// TIA Portal project "TON_VS_P" (V15.1)

(* hardware
DEVICE "S71500/ET200MP station_1"  S7-1500 station
   slot 0: "Rail_0"  Rack  6ES7 590-1***0-0AA0
   slot 1: "PLC_1"  CPU 1513-1 PN  6ES7 513-1AL02-0AB0  V2.6
      slot 3: "CPU display_1"  6ES7591-1AA00-0AA0
DEVICE "HMI_1"  KTP900 Basic PN
   slot 0: "HMI_1"  KTP900 Basic PN  6AV2 123-2JB03-0AX0  15.1.0.0
   slot 1: "HMI_RT_1"  KTP900 Basic PN  6AV2 123-2JB03-0AX0  15.1.0.0
   slot 5: "HMI_1.IE_CP_1"  PROFINET Interface  15.0.1.0
      slot 1: "PROFINET Interface_1"  PROFINET Interface
         slot 1: "Port_1"  Port
*)

// ===== PLC "PLC_1"  CPU 1513-1 PN =====

VAR_GLOBAL   // PLC tag table "Default tag table"
   "Clock_Byte" AT %MB0 : Byte;
   "Clock_10Hz" AT %M0.0 : Bool;
   "Clock_5Hz" AT %M0.1 : Bool;
   "Clock_2.5Hz" AT %M0.2 : Bool;
   "Clock_2Hz" AT %M0.3 : Bool;
   "Clock_1.25Hz" AT %M0.4 : Bool;
   "Clock_1Hz" AT %M0.5 : Bool;
   "Clock_0.625Hz" AT %M0.6 : Bool;
   "Clock_0.5Hz" AT %M0.7 : Bool;
END_VAR

DATA_BLOCK "timer_ore_rfe_DB"   // DB1
{ S7_Optimized_Access := 'TRUE' }
VERSION : 0.1
// stored: InstanceOfName timer_ore_rfe
"timer_ore_rfe"
BEGIN
END_DATA_BLOCK

DATA_BLOCK "timer_ore_ton_DB"   // DB2
{ S7_Optimized_Access := 'TRUE' }
VERSION : 0.1
// stored: InstanceOfName timer_ore_ton
"timer_ore_ton"
BEGIN
END_DATA_BLOCK

DATA_BLOCK "timer_ton"   // DB3
{ S7_Optimized_Access := 'TRUE' }
VERSION : 0.1
   VAR
      btn_reset : Bool;
      permisiune_plecare : Bool;
      terminat : Bool;
      led_pornire : Bool;
      timer_s : Time;
      timer_m : USInt;
      timer_h : USInt;
      timer_s_secunde : Time;
   END_VAR
BEGIN
END_DATA_BLOCK

DATA_BLOCK "timer_rfe"   // DB4
{ S7_Optimized_Access := 'TRUE' }
VERSION : 0.1
   VAR
      btn_reset : Bool;
      permisiune_plecare : Bool;
      terminat : Bool;
      led_pornire : Bool;
      timer_s : USInt;
      timer_m : USInt;
      timer_h : USInt;
   END_VAR
BEGIN
END_DATA_BLOCK

// folder: System blocks/Program resources

DATA_BLOCK "timer_reset_rfe"   // DB5
{ S7_Optimized_Access := 'TRUE' }
AUTHOR : Simatic
FAMILY : IEC
NAME : IEC_TMR
VERSION : 1.0
// stored: InstanceOfName IEC_TIMER
"IEC_TIMER"
BEGIN
END_DATA_BLOCK

DATA_BLOCK "timer_reset_ton"   // DB6
{ S7_Optimized_Access := 'TRUE' }
AUTHOR : Simatic
FAMILY : IEC
NAME : IEC_TMR
VERSION : 1.0
// stored: InstanceOfName IEC_TIMER
"IEC_TIMER"
BEGIN
END_DATA_BLOCK

// folder: (top level)

FUNCTION_BLOCK "timer_ore_rfe"   // FB1, LAD
{ S7_Optimized_Access := 'TRUE' }
VERSION : 0.1
   VAR_INPUT
      reset : Bool;
   END_VAR
   VAR_OUTPUT
      terminat : Bool;
   END_VAR
   VAR_IN_OUT
      permisiune_plecare : Bool;
      timer_s : USInt;
      timer_m : USInt;
      timer_h : USInt;
   END_VAR
   VAR
      re1 : Bool;
   END_VAR
   VAR_TEMP   // added for the SCL form of the ladder/FBD networks
      _w1 : Bool;
   END_VAR
BEGIN

REGION Network 1: timer secunde
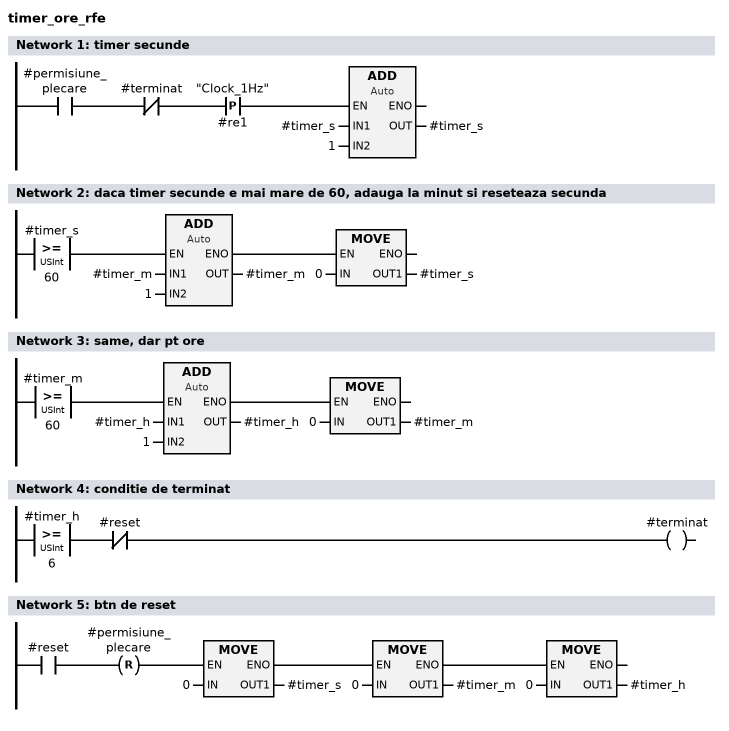
   RUNG wire#powerrail
      Contact( #permisiune_plecare )
      I_Contact( #terminat )
      P_Contact(operand := "Clock_1Hz", bit := #re1)
      Add(in1 := #timer_s, in2 := 1, out => #timer_s)
   END_RUNG
   // the same network as SCL:
   #_w1 := #permisiune_plecare AND NOT #terminat AND "Clock_1Hz" AND NOT #re1;   // rising edge of "Clock_1Hz"
   #re1 := "Clock_1Hz";
   IF #_w1 THEN #timer_s := #timer_s + 1; END_IF;
END_REGION

REGION Network 2: daca timer secunde e mai mare de 60, adauga la minut si reseteaza secunda
   RUNG wire#powerrail
      { S7_Templates := "SrcType := USInt" } GE_Contact(in1 := #timer_s, in2 := 60)
      Add(in1 := #timer_m, in2 := 1, out => #timer_m)
      Move(in := 0, out1 => #timer_s)
   END_RUNG
   // the same network as SCL:
   IF #timer_s >= 60 THEN
       #timer_m := #timer_m + 1;
       #timer_s := 0;
   END_IF;
END_REGION

REGION Network 3: same, dar pt ore
   RUNG wire#powerrail
      { S7_Templates := "SrcType := USInt" } GE_Contact(in1 := #timer_m, in2 := 60)
      Add(in1 := #timer_h, in2 := 1, out => #timer_h)
      Move(in := 0, out1 => #timer_m)
   END_RUNG
   // the same network as SCL:
   IF #timer_m >= 60 THEN
       #timer_h := #timer_h + 1;
       #timer_m := 0;
   END_IF;
END_REGION

REGION Network 4: conditie de terminat
   RUNG wire#powerrail
      { S7_Templates := "SrcType := USInt" } GE_Contact(in1 := #timer_h, in2 := 6)
      I_Contact( #reset )
      Coil( #terminat )
   END_RUNG
   // the same network as SCL:
   #terminat := (#timer_h >= 6) AND NOT #reset;
END_REGION

REGION Network 5: btn de reset
   RUNG wire#powerrail
      Contact( #reset )
      R_Coil( #permisiune_plecare )
      Move(in := 0, out1 => #timer_s)
      Move(in := 0, out1 => #timer_m)
      Move(in := 0, out1 => #timer_h)
   END_RUNG
   // the same network as SCL:
   IF #reset THEN
       #permisiune_plecare := FALSE;
       #timer_s := 0;
       #timer_m := 0;
       #timer_h := 0;
   END_IF;
END_REGION
END_FUNCTION_BLOCK

FUNCTION_BLOCK "timer_ore_ton"   // FB2, LAD
TITLE = aceasta functie nu prea o sa aiba sens, but bare with me ig
{ S7_Optimized_Access := 'TRUE' }
VERSION : 0.1
   VAR_INPUT
      reset : Bool;
   END_VAR
   VAR_OUTPUT
      terminat : Bool;
   END_VAR
   VAR_IN_OUT
      permisiune_plecare : Bool;
      time_ore : USInt;
      time_min : USInt;
      time_sec : Time;
   END_VAR
   VAR
      ton_s : TON_TIME;
      ton_aux : TON_TIME;
      terminat_secunde : Bool;
      plecare_sec : Bool;
      plecare_min : Bool;
      re1 : Bool;
      plecare_ora : Bool;
      adaugat_minut : Bool;
   END_VAR
   VAR_TEMP   // added for the SCL form of the ladder/FBD networks
      _w1 : Bool;
   END_VAR
BEGIN

REGION Network 1
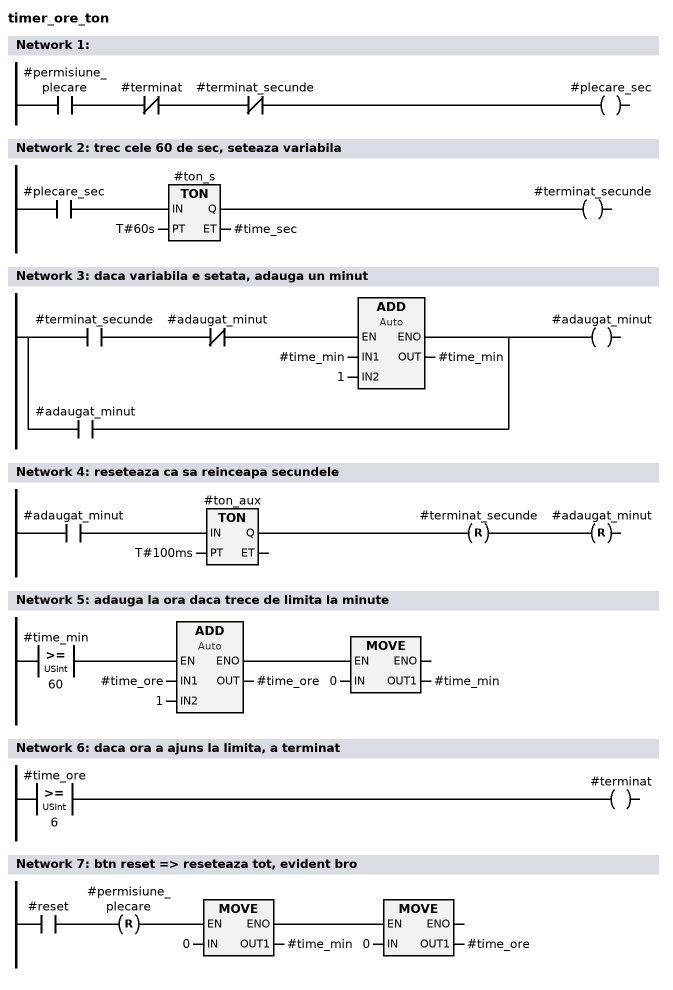
   RUNG wire#powerrail
      Contact( #permisiune_plecare )
      I_Contact( #terminat )
      I_Contact( #terminat_secunde )
      Coil( #plecare_sec )
   END_RUNG
   // the same network as SCL:
   #plecare_sec := #permisiune_plecare AND NOT #terminat AND NOT #terminat_secunde;
END_REGION

REGION Network 2: trec cele 60 de sec, seteaza variabila
   #ton_s(IN := #plecare_sec, PT := T#60s, ET => #time_sec);   // TON
   #terminat_secunde := #ton_s.Q;
END_REGION

REGION Network 3: daca variabila e setata, adauga un minut
   RUNG wire#powerrail
      Contact( #terminat_secunde )
      I_Contact( #adaugat_minut )
      Add(in1 := #time_min, in2 := 1, out => #time_min)
      wire#w1
      Coil( #adaugat_minut )
   END_RUNG
   RUNG wire#powerrail
      Contact( #adaugat_minut )
   END_RUNG wire#w1
   // the same network as SCL:
   #_w1 := #terminat_secunde AND NOT #adaugat_minut;
   IF #_w1 THEN #time_min := #time_min + 1; END_IF;
   #adaugat_minut := #_w1 OR #adaugat_minut;
END_REGION

REGION Network 4: reseteaza ca sa reinceapa secundele
   #ton_aux(IN := #adaugat_minut, PT := T#100ms);   // TON
   IF #ton_aux.Q THEN
       #terminat_secunde := FALSE;
       #adaugat_minut := FALSE;
   END_IF;
END_REGION

REGION Network 5: adauga la ora daca trece de limita la minute
   RUNG wire#powerrail
      { S7_Templates := "SrcType := USInt" } GE_Contact(in1 := #time_min, in2 := 60)
      Add(in1 := #time_ore, in2 := 1, out => #time_ore)
      Move(in := 0, out1 => #time_min)
   END_RUNG
   // the same network as SCL:
   IF #time_min >= 60 THEN
       #time_ore := #time_ore + 1;
       #time_min := 0;
   END_IF;
END_REGION

REGION Network 6: daca ora a ajuns la limita, a terminat
   RUNG wire#powerrail
      { S7_Templates := "SrcType := USInt" } GE_Contact(in1 := #time_ore, in2 := 6)
      Coil( #terminat )
   END_RUNG
   // the same network as SCL:
   #terminat := #time_ore >= 6;
END_REGION

REGION Network 7: btn reset => reseteaza tot, evident bro
   RUNG wire#powerrail
      Contact( #reset )
      R_Coil( #permisiune_plecare )
      Move(in := 0, out1 => #time_min)
      Move(in := 0, out1 => #time_ore)
   END_RUNG
   // the same network as SCL:
   IF #reset THEN
       #permisiune_plecare := FALSE;
       #time_min := 0;
       #time_ore := 0;
   END_IF;
END_REGION
END_FUNCTION_BLOCK

ORGANIZATION_BLOCK "Main"   // OB1, LAD, ProgramCycle
TITLE = "Main Program Sweep (Cycle)"
{ S7_Optimized_Access := 'TRUE' }
VERSION : 0.1
   VAR_INPUT
      Initial_Call : Bool;   // Initial call of this OB
      Remanence : Bool;   // =True, if remanent data are available
   END_VAR
BEGIN

REGION Network 1: functii
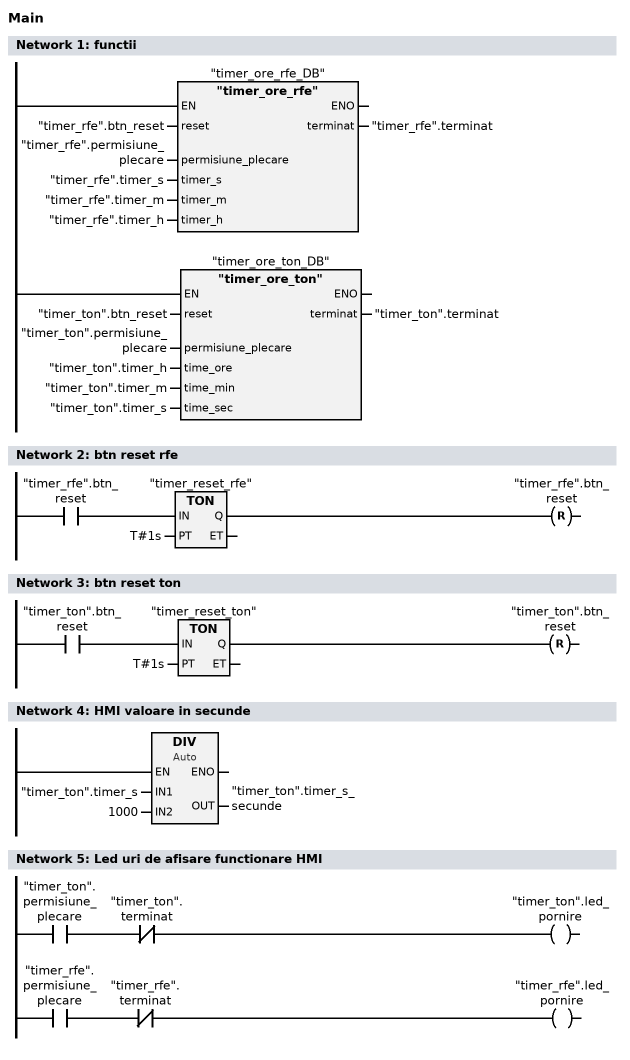
   RUNG wire#powerrail
      "timer_ore_rfe_DB"(reset := "timer_rfe".btn_reset, permisiune_plecare := "timer_rfe".permisiune_plecare, timer_s := "timer_rfe".timer_s, timer_m := "timer_rfe".timer_m, timer_h := "timer_rfe".timer_h, terminat => "timer_rfe".terminat)
   END_RUNG
   RUNG wire#powerrail
      "timer_ore_ton_DB"(reset := "timer_ton".btn_reset, permisiune_plecare := "timer_ton".permisiune_plecare, time_ore := "timer_ton".timer_h, time_min := "timer_ton".timer_m, time_sec := "timer_ton".timer_s, terminat => "timer_ton".terminat)
   END_RUNG
   // the same network as SCL:
   "timer_ore_rfe_DB"(reset := "timer_rfe".btn_reset,   // "timer_ore_rfe"
                      permisiune_plecare := "timer_rfe".permisiune_plecare,
                      timer_s := "timer_rfe".timer_s,
                      timer_m := "timer_rfe".timer_m,
                      timer_h := "timer_rfe".timer_h,
                      terminat => "timer_rfe".terminat);
   "timer_ore_ton_DB"(reset := "timer_ton".btn_reset,   // "timer_ore_ton"
                      permisiune_plecare := "timer_ton".permisiune_plecare,
                      time_ore := "timer_ton".timer_h,
                      time_min := "timer_ton".timer_m,
                      time_sec := "timer_ton".timer_s,
                      terminat => "timer_ton".terminat);
END_REGION

REGION Network 2: btn reset rfe
   "timer_reset_rfe".TON(IN := "timer_rfe".btn_reset, PT := T#1s);
   IF "timer_reset_rfe".Q THEN "timer_rfe".btn_reset := FALSE; END_IF;
END_REGION

REGION Network 3: btn reset ton
   "timer_reset_ton".TON(IN := "timer_ton".btn_reset, PT := T#1s);
   IF "timer_reset_ton".Q THEN "timer_ton".btn_reset := FALSE; END_IF;
END_REGION

REGION Network 4: HMI valoare in secunde
   RUNG wire#powerrail
      Div(in1 := "timer_ton".timer_s, in2 := 1000, out => "timer_ton".timer_s_secunde)
   END_RUNG
   // the same network as SCL:
   "timer_ton".timer_s_secunde := "timer_ton".timer_s / 1000;
END_REGION

REGION Network 5: Led uri de afisare functionare HMI
   RUNG wire#powerrail
      Contact( "timer_ton".permisiune_plecare )
      I_Contact( "timer_ton".terminat )
      Coil( "timer_ton".led_pornire )
   END_RUNG
   RUNG wire#powerrail
      Contact( "timer_rfe".permisiune_plecare )
      I_Contact( "timer_rfe".terminat )
      Coil( "timer_rfe".led_pornire )
   END_RUNG
   // the same network as SCL:
   "timer_ton".led_pornire := "timer_ton".permisiune_plecare AND NOT "timer_ton".terminat;
   "timer_rfe".led_pornire := "timer_rfe".permisiune_plecare AND NOT "timer_rfe".terminat;
END_REGION
END_ORGANIZATION_BLOCK

(* ===== HMI "HMI_RT_1" =====
system functions are stored by id; their names below are inferred from use
connection "HMI_Connection_1": ETHERNET, SMART_S7_1500_OMS

HMI tags "Default tag table"
   "timer_ton_timer_s" : Time = PLC timer_ton.timer_s, 1 s
   "timer_ton_timer_m" : USInt = PLC timer_ton.timer_m, 1 s
   "timer_ton_timer_h" : USInt = PLC timer_ton.timer_h, 1 s
   "timer_ton_terminat" : Bool = PLC timer_ton.terminat, 1 s
   "timer_ton_btn_reset" : Bool = PLC timer_ton.btn_reset, 1 s
   "timer_rfe_btn_reset" : Bool = PLC timer_rfe.btn_reset, 1 s
   "timer_rfe_terminat" : Bool = PLC timer_rfe.terminat, 1 s
   "timer_rfe_timer_s" : USInt = PLC timer_rfe.timer_s, 1 s
   "timer_rfe_timer_m" : USInt = PLC timer_rfe.timer_m, 1 s
   "timer_rfe_timer_h" : USInt = PLC timer_rfe.timer_h, 1 s
   "timer_ton_permisiune_plecare" : Bool = PLC timer_ton.permisiune_plecare, 1 s
   "timer_rfe_permisiune_plecare" : Bool = PLC timer_rfe.permisiune_plecare, 1 s
   "timer_ton_timer_s_secunde" : Time = PLC timer_ton.timer_s_secunde, 1 s
   "timer_rfe_led_pornire" : Bool = PLC timer_rfe.led_pornire, 1 s
   "timer_ton_led_pornire" : Bool = PLC timer_ton.led_pornire, 1 s

Template "Template_1" 800x480
   Button "Exit" at 722,440 size 55x39; TextOff 'Exit'; PictureOff "ExitRuntime_KTP900_Basic_PN_TR"; PictureOn "ExitRuntime_KTP900_Basic_PN_TR"
      on Release: StopRuntime(0)
   Button "Start screen" at 22,440 size 55x39; TextOff 'Start screen'; PictureOff "NavigateHome_KTP900_Basic_PN_TR"; PictureOn "NavigateHome_KTP900_Basic_PN_TR"
      on Release: ActivateScreen("Simulare", 0)

screen "Simulare" 800x480, template "Template_1"
   TextField "Text field_1" at 157,22 size 94x25; Text 'Timer TON'
   TextField "Text field_2" at 572,22 size 90x25; Text 'Timer RFE'
   IOField "I/O field_1" at 39,152 size 54x32; FormatPattern 999; Unit s
      ProcessValue <- "timer_ton_timer_s_secunde"
   IOField "I/O field_2" at 39,228 size 54x32; FormatPattern 999; Unit m
      ProcessValue <- "timer_ton_timer_m"
   IOField "I/O field_3" at 39,310 size 54x32; FormatPattern 999; Unit h
      ProcessValue <- "timer_ton_timer_h"
   Button "Button_1" at 193,227 size 96x32; TextOff 'Reset'
      on Click: SetBit("timer_ton_btn_reset")
   Circle "Circle_1" at 219,307 size 48x48
      Appearance <- "timer_ton_terminat"
   TextField "Text field_3" at 212,277 size 62x20; Text 'Terminat'
   IOField "I/O field_4" at 464,152 size 54x32; FormatPattern 999; Unit s
      ProcessValue <- "timer_rfe_timer_s"
   IOField "I/O field_5" at 464,228 size 54x32; FormatPattern 999; Unit m
      ProcessValue <- "timer_rfe_timer_m"
   IOField "I/O field_6" at 464,310 size 54x32; FormatPattern 999; Unit h
      ProcessValue <- "timer_rfe_timer_h"
   Button "Button_2" at 618,227 size 96x32; TextOff 'Reset'
      on Click: SetBit("timer_rfe_btn_reset")
   Circle "Circle_2" at 644,307 size 48x48
      Appearance <- "timer_rfe_terminat"
   TextField "Text field_4" at 637,277 size 62x20; Text 'Terminat'
   Button "Button_3" at 193,163 size 96x32; TextOff 'Pornire'
      on Click: SetBit("timer_ton_permisiune_plecare")
   Button "Button_4" at 619,163 size 96x32; TextOff 'Pornire'
      on Click: SetBit("timer_rfe_permisiune_plecare")
   Circle "Circle_3" at 127,100 size 48x48
      Appearance <- "timer_ton_led_pornire"
   TextField "Text field_5" at 129,72 size 44x20; Text 'Pornit'
   Circle "Circle_4" at 547,100 size 48x48
      Appearance <- "timer_rfe_led_pornire"
   TextField "Text field_6" at 549,72 size 44x20; Text 'Pornit'
*)